{attribute 'GeneratedUsingTerminal: EP9128-0021-0019'}
{attribute addProperty BoxType "EP9128-0021-0019"}
{attribute addProperty Id "A_0016_EP9214_0023_0019EP9214_4599284580A_0017_EP9214_0023_0020EP9214_4599284580A_0018_EP9214_0023_0021EP9214_4599284580A_0019_EP9214_0023_0022EP9214_4599284580A_0020_EP9224_0023_0016EP9224_1EB2867A112A_0021_EP9224_0023_0017EP9224_1EB2867A112A_0024_EP9521_0020_0000A_0024_EP9521_0020_0000_16465A9C29A_0022_EP9224_0037_0017A_0022_EP9224_0037_0017_201EEDCE2A_0013_EP9128_0021_0019_2_EP9128_1021EP9128_AB5A94672A_0013_EP9128_0021_0019_3_EP9128_2021EP9128_AB5A94672"}
{attribute addProperty CRC "2673461629"}
{attribute addProperty Size "579"}
TYPE A_0013_EP9128_0021_0019_9F59C97D EXTENDS EP9128_AB5A9467 :
STRUCT
	{attribute addProperty Name "A_0016_EP9214_0023_0019"}
	{attribute addProperty PreviousPort "A_0013(EP9128-0021-0019) : D"}
	A_0016_EP9214_0023_0019 : EP9214_45992845;
	{attribute addProperty Name "A_0017_EP9214_0023_0020"}
	{attribute addProperty PreviousPort "A_0016(EP9214-0023-0019) : B"}
	A_0017_EP9214_0023_0020 : EP9214_45992845;
	{attribute addProperty Name "A_0018_EP9214_0023_0021"}
	{attribute addProperty PreviousPort "A_0017(EP9214-0023-0020) : B"}
	A_0018_EP9214_0023_0021 : EP9214_45992845;
	{attribute addProperty Name "A_0019_EP9214_0023_0022"}
	{attribute addProperty PreviousPort "A_0018(EP9214-0023-0021) : B"}
	A_0019_EP9214_0023_0022 : EP9214_45992845;
	{attribute addProperty Name "A_0020_EP9224_0023_0016"}
	{attribute addProperty PreviousPort "A_0019(EP9214-0023-0022) : B"}
	A_0020_EP9224_0023_0016 : EP9224_1EB2867A;
	{attribute addProperty Name "A_0021_EP9224_0023_0017"}
	{attribute addProperty PreviousPort "A_0020(EP9224-0023-0016) : B"}
	A_0021_EP9224_0023_0017 : EP9224_1EB2867A;
	{attribute addProperty Name "A_0024_EP9521_0020_0000"}
	{attribute addProperty PreviousPort "A_0021(EP9224-0023-0017) : B"}
	A_0024_EP9521_0020_0000 : A_0024_EP9521_0020_0000_16465A9C;
	{attribute addProperty Name "A_0022_EP9224_0037_0017"}
	{attribute addProperty PreviousPort "A_0024(EP9521-0020-0000) : C"}
	A_0022_EP9224_0037_0017 : A_0022_EP9224_0037_0017_201EEDCE;
	{attribute addProperty Name "A_0013_EP9128_0021_0019_2_EP9128_1021"}
	{attribute addProperty PreviousPort "A_0013(EP9128-0021-0019) : C"}
	A_0013_EP9128_0021_0019_2_EP9128_1021 : EP9128_AB5A9467;
	{attribute addProperty Name "A_0013_EP9128_0021_0019_3_EP9128_2021"}
	{attribute addProperty PreviousPort "A_0013(EP9128-0021-0019)_2 (EP9128-1021) : C"}
	A_0013_EP9128_0021_0019_3_EP9128_2021 : EP9128_AB5A9467;
END_STRUCT
END_TYPE

(* stored: Version 1.2.0.0, ProductVersion 3.1.4024.9
   DUT A_0013_EP9128_0021_0019_9F59C97D: Id {891532e9-8feb-48dc-b8e8-026089aad436} *)
